// TIA Portal V16 export
// export: Created 2021-08-04T22:56:06.8663411Z, ExportSetting WithDefaults, DisplayName Totally Integrated Automation Portal, DisplayVersion V16 Update 4, DisplayName TIA Portal Version Control Interface, DisplayVersion V16 Update 2, DisplayName TIA Portal Openness, DisplayVersion V16 Update 4, DisplayName STEP 7 Professional, DisplayVersion V16 Update 4, DisplayName STEP 7 Safety, DisplayVersion V16, DisplayName WinCC Advanced, DisplayVersion V16 Update 4
FUNCTION_BLOCK "BlockIncrementer"   // FB3, F_FBD
{ S7_Optimized_Access := 'TRUE' }
VERSION : 0.1
// stored: AutoNumber true, IsIECCheckEnabled false, UDAEnableTagReadback false
   VAR
      "a" : "MyCounter";
      "b" : "MyCounter";
   END_VAR
BEGIN

REGION Network 1
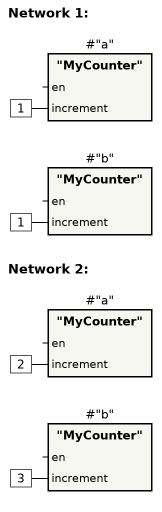
   #"a"(increment := 1);   // "MyCounter"
   #"b"(increment := 1);   // "MyCounter"
END_REGION

REGION Network 2
   #"a"(increment := 2);   // "MyCounter"
   #"b"(increment := 3);   // "MyCounter"
END_REGION
END_FUNCTION_BLOCK
